# EPICS autosave request: iocBoot/ioc13Keithley2/auto_settings.req
file "Keithley2kDMM_mf22_settings.req", P=$(P), Dmm=DMM1
file "pid_control_settings.req"         P=$(P), PID=PID1
file "scan_settings.req",               P=$(P), S=scan1
file "scan_settings.req",               P=$(P), S=scan2
file "scan_settings.req",               P=$(P), S=scan3
file "scan_settings.req",               P=$(P), S=scan4
